{attribute 'GeneratedUsingTerminal: EK1100-0000-0018'}
{attribute addProperty BoxType "EK1100-0000-0018"}
{attribute addProperty Id "Beckhoff_ER7xxxEK1122Beckhoff_ER7xxxEK1122_C13D679B598"}
{attribute addProperty CRC "1548888022"}
{attribute addProperty Size "598"}
TYPE Beckhoff_ER7xxx_5C5227D6 EXTENDS EK1100_1FC0878B :
STRUCT
	{attribute addProperty Name "Beckhoff_ER7xxxEK1122"}
	{attribute addProperty PreviousPort "Beckhoff ER7xxx : B"}
	Beckhoff_ER7xxxEK1122 : Beckhoff_ER7xxxEK1122_C13D679B;
END_STRUCT
END_TYPE

(* stored: Version 1.2.0.0, ProductVersion 3.1.4024.9
   DUT Beckhoff_ER7xxx_5C5227D6: Id {66fc5b6c-a2c2-4c7e-9c10-79bb59b4faed} *)
